Fanuc KAREL source: kt00935.KL

-- PROVISIONAL review KL for V1013-1; original PC SHA256 85cd03b5a56e0ae309ade5c14cb749353b7afb776ee1fd3d91e5fc99c4d270b8
-- Incomplete behavior may be omitted. Consult companion uncertainty JSON. Do not deploy.
PROGRAM KT00935
%NOLOCKGROUP
VAR
  ENTRY : INTEGER
  PNAME : STRING[80]
  VNAME : STRING[80]
  STATUS : INTEGER
  VALUE : BOOLEAN
BEGIN
  -- UNRESOLVED_PC offsets 5-12; opcodes 9C,23
  -- UNRESOLVED_PC offsets 17-25; opcodes 3F,75
  -- UNRESOLVED_PC offsets 30-43; opcodes 3F,75
  -- UNRESOLVED_PC offsets 48-86; opcodes 27,22,22,2A,22,2A,22,22,AF
  -- UNRESOLVED_PC offsets 91-95; opcodes 7F
END KT00935
